{attribute addProperty BoxType "EL9560-0000-0016"}
{attribute addProperty Id "Status_UsAT %I*Status_Us_324A4102810Status_UoAT %I*Status_Uo_324A4102810WcStateAT %I*WcState_98A4DF7520.250InfoDataAT %I*InfoData_192954DE1620"}
{attribute addProperty CRC "37654351"}
{attribute addProperty SizeInBites "34"}
{attribute addProperty SizeInBytes "4.25"}
TYPE EL9560_84A42FC9 :
STRUCT
	{attribute addProperty Name "Status_Us"}
	Status_Us : Status_Us_324A4102;
	{attribute addProperty Name "Status_Uo"}
	Status_Uo : Status_Uo_324A4102;
	{attribute addProperty Name "WcState"}
	WcState : WcState_98A4DF75;
	{attribute addProperty Name "InfoData"}
	InfoData : InfoData_192954DE;
END_STRUCT
END_TYPE

(* stored: Version 1.2.0.0, ProductVersion 3.1.4024.9
   DUT EL9560_84A42FC9: Id {fb10d2cb-cd42-4e28-b2d8-521154af9119} *)
